VAR_GLOBAL
		bTest			: BOOL;
		nTest			: INT;
		rlTest			: REAL;
		stTest			: ST_PyADS_Test;
END_VAR

(* stored: Version 1.1.0.1, ProductVersion 3.1.4024.12
   GVL GVL_Ads: Id {7e362bda-4518-4d8c-953b-2044b03a7bff} *)
